{attribute 'GeneratedUsingTerminal: EJ2918-0000-0017'}
{attribute addProperty BoxType "EJ2918-0000-0017"}
{attribute addProperty Id "FSOEAT %I*FSOE_046F804E7"}
{attribute addProperty CRC "2476392253"}
{attribute addProperty Size "7"}
TYPE FSoE_Inputs_939ABF3D :
STRUCT
	{attribute addProperty Name "FSOE"}
	FSOE AT %I* : FSOE_046F804E;
END_STRUCT
END_TYPE

(* stored: Version 1.2.0.0, ProductVersion 3.1.4024.9
   DUT FSoE_Inputs_939ABF3D: Id {49385fa6-10ba-4fae-9df2-b0dc345a3ae0} *)
